// TIA Portal V20 export
TYPE "CommonPartData"
// stored: Access Published
   STRUCT
      PartType : Byte;
      PartStatus1 : Byte;
      PartStatus2 : Byte;
      LastMachineNumber : Byte;
      ProductionTimestamp : DTL;   // TimeStamp
      Part_ID : String[32];
   END_STRUCT;
END_TYPE
